{attribute addProperty BoxType "EP2316-0008-0017"}
{attribute addProperty Id "DO_Diag_InputsAT %I*DO_Diag_Inputs_9F71B9E27290DO_Diag_Inputs_1AT %I*DO_Diag_Inputs_8D5DE8777290DO_Inputs_DeviceAT %I*DO_Inputs_Device_BB3041553240DO_OutputsAT %Q*DO_Outputs_33B763766480DO_Outputs_DeviceAT %Q*DO_Outputs_Device_735003021620WcStateAT %I*WcState_F855686C1620InfoDataAT %I*InfoData_BC63D37F80100"}
{attribute addProperty CRC "1870889898"}
{attribute addProperty SizeInBites "352"}
{attribute addProperty SizeInBytes "44"}
TYPE EP2316_900F0E4A :
STRUCT
	{attribute addProperty Name "DO_Diag_Inputs"}
	DO_Diag_Inputs : DO_Diag_Inputs_9F71B9E2;
	{attribute addProperty Name "DO_Diag_Inputs_1"}
	DO_Diag_Inputs_1 : DO_Diag_Inputs_8D5DE877;
	{attribute addProperty Name "DO_Inputs_Device"}
	DO_Inputs_Device : DO_Inputs_Device_BB304155;
	{attribute addProperty Name "DO_Outputs"}
	DO_Outputs : DO_Outputs_33B76376;
	{attribute addProperty Name "DO_Outputs_Device"}
	DO_Outputs_Device : DO_Outputs_Device_73500302;
	{attribute addProperty Name "WcState"}
	WcState : WcState_F855686C;
	{attribute addProperty Name "InfoData"}
	InfoData : InfoData_BC63D37F;
END_STRUCT
END_TYPE

(* stored: Version 1.2.0.0, ProductVersion 3.1.4024.9
   DUT EP2316_900F0E4A: Id {7f7b5b95-1ed7-4110-9372-6c2f0af87fb3} *)
